TYPE st_TCME31_Set :
STRUCT
	IPAddress		:	String := '192.168.1.70';
	
	DigitalOutput1	:	Bool;
	DigitalOutput2	:	Bool;
	DigitalOutput3	:	Bool;
	DigitalOutput4	:	Bool;
END_STRUCT
END_TYPE

(* stored: Version 1.1.0.1, ProductVersion 3.1.4026.18
   DUT st_TCME31_Set: Id {2cdec817-d5ed-4bf9-b8af-d8cf72a78442} *)
